TYPE TcoEntityBase EXTENDS TcoData.TcoEntity :
STRUCT
	{attribute clr [RenderIgnore("Control", "ShadowControl")]}
	{attribute addProperty Name "<#Created#>"}
	_Created : DT;
	{attribute clr [RenderIgnore("Control", "ShadowControl")]}
	{attribute addProperty Name "<#Modified#>"}
	_Modified : DT;
	
END_STRUCT
END_TYPE

(* stored: Version 1.1.0.1
   DUT TcoEntityBase: Id {c8c4cc6f-61a4-4ead-b300-8aa0513c06f9} *)
